// SIMATIC S7-200 project (STEP 7-Micro/WIN), CPU 226 CN REL 02.01

ORGANIZATION_BLOCK 主程序:OB1
TITLE=程序注释
BEGIN
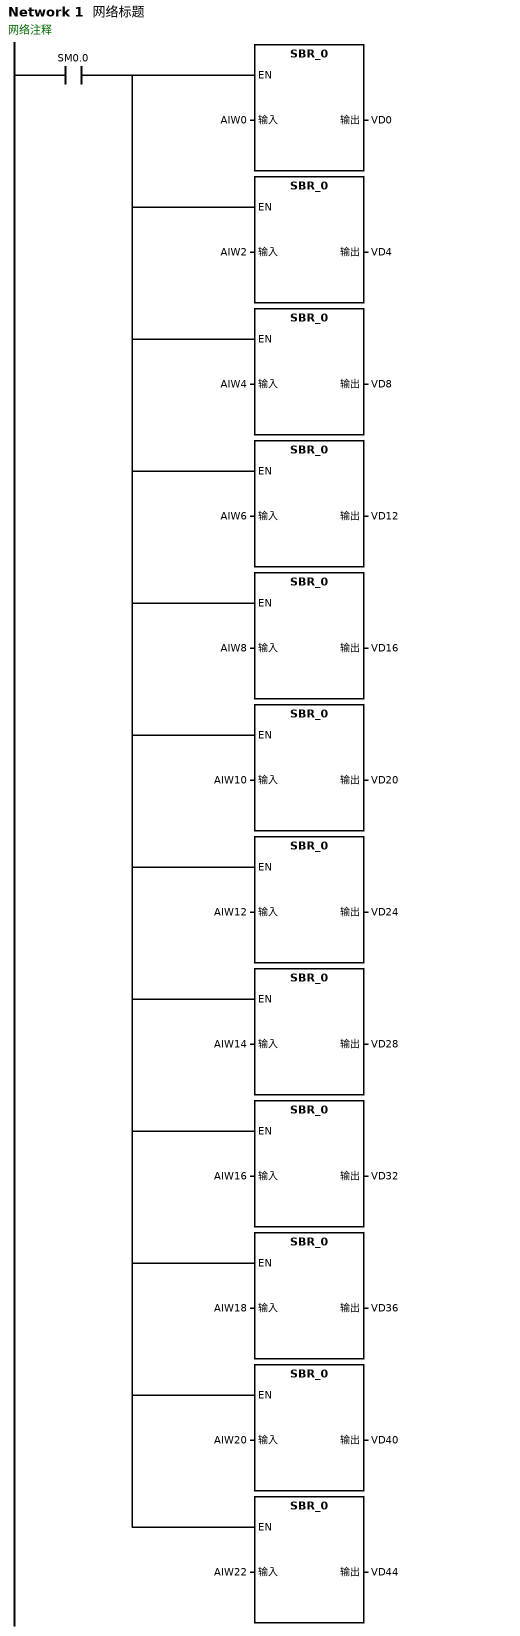
Network 1 // 网络标题
// 网络注释
LD     SM0.0
CALL   SBR_0:SBR0, AIW0, VD0
CALL   SBR_0:SBR0, AIW2, VD4
CALL   SBR_0:SBR0, AIW4, VD8
CALL   SBR_0:SBR0, AIW6, VD12
CALL   SBR_0:SBR0, AIW8, VD16
CALL   SBR_0:SBR0, AIW10, VD20
CALL   SBR_0:SBR0, AIW12, VD24
CALL   SBR_0:SBR0, AIW14, VD28
CALL   SBR_0:SBR0, AIW16, VD32
CALL   SBR_0:SBR0, AIW18, VD36
CALL   SBR_0:SBR0, AIW20, VD40
CALL   SBR_0:SBR0, AIW22, VD44
END_ORGANIZATION_BLOCK

SUBROUTINE_BLOCK SBR_0:SBR0
TITLE=子程序注释
VAR_INPUT
输入:INT;	// LW0 
END_VAR
VAR_OUTPUT
输出:REAL;	// LD2 
END_VAR
BEGIN
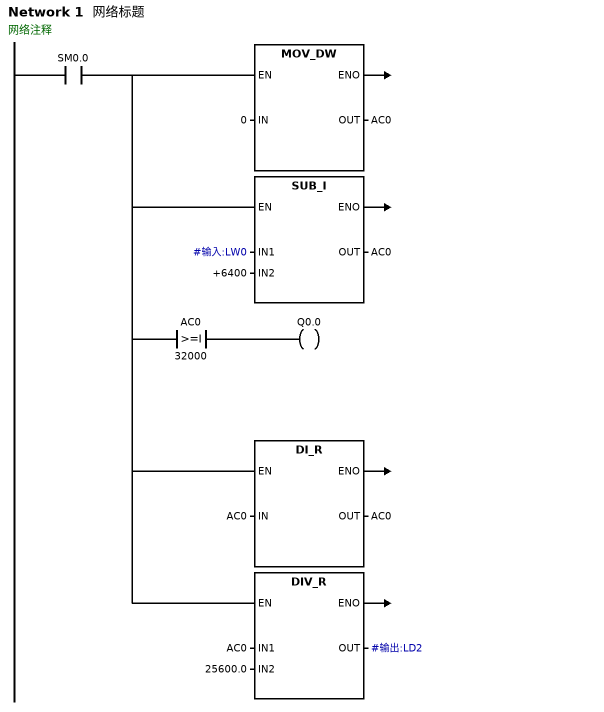
Network 1 // 网络标题
// 网络注释
// (network saved uncompiled; LAD cells follow)
// row 0: c0 -| |- SM0.0 v  c1 --  c2 [MOV_DW EN:=power@row0, IN:=0, ENO=>power, OUT=>AC0]  c3 ->
// row 1: c0 ^v  c2 [box]
// row 2: c0 ^v  c1 --  c2 [SUB_I EN:=power@row2, IN1:=#输入:LW0, IN2:=+6400, ENO=>power, OUT=>AC0]  c3 ->
// row 3: c0 ^v  c2 [box]
// row 4: c0 ^v  c1 -|>=I|- AC0, 32000  c2 -( ) Q0.0
// row 5: c0 ^v
// row 6: c0 ^v  c1 --  c2 [DI_R EN:=power@row6, IN:=AC0, ENO=>power, OUT=>AC0]  c3 ->
// row 7: c0 ^v  c2 [box]
// row 8: c0 ^  c1 --  c2 [DIV_R EN:=power@row8, IN1:=AC0, IN2:=25600.0, ENO=>power, OUT=>#输出:LD2]  c3 ->
// row 9: c2 [box]
END_SUBROUTINE_BLOCK
